SUBAPPLICATION Uebung_201_AX (* Interlock: ILOCK_BLOCK_AX (Gegenseitige Verriegelung via Adapter) *)
  (* Standard: 61499-2; Description: Copyright (c) 2023 Meisterschulen am Ostbahnhof This program and the accompanying materials are made available under the terms of the Eclipse Public License 2.0 which is available at https://www.eclipse.org/legal/epl-2.0/ SPDX-License-Identifier: EPL-2.0 *)
  (* Version 1.0, 2026-04-19, Franz Höpfinger, Meisterschulen am Ostbahnhof, initial API and implementation and/or initial documentation *)
  PACKAGE Uebungen;
  IMPORT logiBUS::io::DI::logiBUS_DI::Input_I1;
  IMPORT logiBUS::io::DI::logiBUS_DI::Input_I2;
  IMPORT logiBUS::io::DQ::logiBUS_DO::Output_Q1;
  IMPORT logiBUS::io::DQ::logiBUS_DO::Output_Q2;
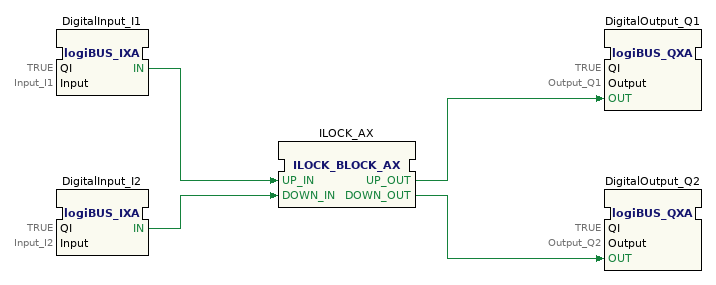
  FBS
    DigitalInput_I1 : logiBUS::io::DI::logiBUS_IXA(QI := TRUE, Input := Input_I1);
    DigitalInput_I2 : logiBUS::io::DI::logiBUS_IXA(QI := TRUE, Input := Input_I2);
    ILOCK_AX : logiBUS::signalprocessing::interlock::ILOCK_BLOCK_AX;
    DigitalOutput_Q1 : logiBUS::io::DQ::logiBUS_QXA(QI := TRUE, Output := Output_Q1);
    DigitalOutput_Q2 : logiBUS::io::DQ::logiBUS_QXA(QI := TRUE, Output := Output_Q2);
  END_FBS
  ADAPTER_CONNECTIONS
    DigitalInput_I1.IN TO ILOCK_AX.UP_IN;
    DigitalInput_I2.IN TO ILOCK_AX.DOWN_IN;
    ILOCK_AX.UP_OUT TO DigitalOutput_Q1.OUT;
    ILOCK_AX.DOWN_OUT TO DigitalOutput_Q2.OUT;
  END_CONNECTIONS
END_SUBAPPLICATION
